(* Log/debug/error message fifo *)
FUNCTION_BLOCK FB_LogFifo
VAR_INPUT
    bLog    : BOOL   := FALSE; (* TRUE => Enable log message output, FALSE => Disable *)
    sPrefix : STRING := 'Unknown::'; (* Log message description string (allows the identification of log message source) *)

    sMessage : STRING := ''; (* String message to add (write) to the fifo *)
    nErrID   : UDINT  := 0; (* Error code to add (write) to the fifo *)
    hSocket  : T_HSOCKET; (* Socket connection handle *)
END_VAR

VAR_OUTPUT
    bOk    : BOOL; (* TRUE = New entry added or removed succesfully, FALSE = Fifo overflow or fifo empty *)
    sGet   : STRING[1000]; (* String entry removed (read) from fifo *)
    nCount : UDINT := 0; (* Number of fifo entries *)
END_VAR

VAR
    fbBuffer : FB_StringRingBuffer; (* Basic (lower level) string buffer control function block *)
    buffer   : ARRAY[0..PLCPRJ_BUFFER_SIZE] OF BYTE; (* Internal buffer memory *)
    sSource  : STRING[1000];
    sPut     : STRING[1000];
END_VAR

;

ACTION Clear:
(* Clears all fifo entries *)
fbBuffer.A_Reset(pBuffer := ADR(buffer), cbBuffer := SIZEOF(buffer), bOk => bOk, nCount => nCount, getValue => sGet);
END_ACTION

ACTION Error:
(* Adds new fifo entry *)
IF nErrID = 0 THEN
    sSource := '::Error: 0x';
ELSIF (nErrID AND 16#80000000) = 16#80000000 THEN
    IF nErrID = 16#80072746 THEN
        sSource := '::Win32 error (the connection is reset by remote side): 0x';
    ELSE
        sSource := '::Win32 error: 0x';
    END_IF
ELSIF (nErrID AND 16#00008100) = 16#00008100 THEN
    CASE nErrID OF
        PLCPRJ_ERROR_RECEIVE_TIMEOUT:
            sSource := '::PLC sample project receive timeout error: 0x';

        PLCPRJ_ERROR_SENDFIFO_OVERFLOW:
            sSource := '::PLC sample project send fifo overflow error: 0x';

        PLCPRJ_ERROR_RECFIFO_OVERFLOW:
            sSource := '::PLC sample project receive fifo overflow error: 0x';

    ELSE
        sSource := '::Other PLC sample project error: 0x';
    END_CASE
ELSIF (nErrID AND 16#00008000) = 16#00008000 THEN
    sSource := '::Internal TCP/IP Connection Server error: 0x';
ELSE
    sSource := '::TwinCAT System error: 0x';
END_IF

sPut := CONCAT(CONCAT(CONCAT(sPrefix, sMessage), sSource), DWORD_TO_HEXSTR(nErrID AND 16#FFFF, 0, FALSE));

fbBuffer.A_AddTail(pBuffer := ADR(buffer), cbBuffer := SIZEOF(buffer), putValue := sPut, bOk => bOk, nCount => nCount);

IF bOk THEN
    IF bLog THEN (* Log error message *)
        ADSLOGSTR(ADSLOG_MSGTYPE_ERROR OR ADSLOG_MSGTYPE_LOG, '%s', sPut);
    END_IF
END_IF
END_ACTION

ACTION Message:
(* Adds new fifo entry *)
sPut := CONCAT(CONCAT(sPrefix, sMessage), CONCAT('::', HSOCKET_TO_STRING(hSocket)));
fbBuffer.A_AddTail(pBuffer := ADR(buffer), cbBuffer := SIZEOF(buffer), putValue := sPut, bOk => bOk, nCount => nCount);

IF bOk THEN
    IF bLog THEN (* Log information message *)
        ADSLOGSTR(ADSLOG_MSGTYPE_HINT OR ADSLOG_MSGTYPE_LOG, '%s', sPut);
    END_IF
END_IF
END_ACTION

ACTION Remove:
(* Removes oldest fifo entry *)
IF nCount = 0 THEN
    sGet := '';
    bOk  := FALSE;
    RETURN;
END_IF

fbBuffer.A_RemoveHead(pBuffer := ADR(buffer), cbBuffer := SIZEOF(buffer), getValue => sGet, bOk => bOk, nCount => nCount);
END_ACTION

END_FUNCTION_BLOCK

(* stored: Version 1.1.0.1
   POU FB_LogFifo: Id {fe866cb2-776b-4698-90f3-99df925c977e}, SpecialFunc None
   Action Clear: Id {ef736a9d-5f3f-48ba-acf6-4d777badc116}
   Action Error: Id {712aac61-775c-47bc-8dac-a1a0cac3c8d9}
   Action Message: Id {f4165a9b-3feb-4a87-ac4d-99ff3481c50e}
   Action Remove: Id {d2c38e3b-ab38-41db-954c-e91c59adbfb9} *)
